{attribute 'hide'}
PROGRAM MAIN
VAR
END_VAR

{IF defined(TEST)}
MAIN_TEST();
{END_IF}

END_PROGRAM

(* stored: Version 1.1.0.1, ProductVersion 3.1.4022.18
   POU MAIN: Id {2c89e8f7-6dea-4729-ad74-2566660fc32d}, SpecialFunc None *)
